DATA_BLOCK "SwitchPLC_Hmi"
{ S7_Optimized_Access := 'TRUE' }
VERSION : 0.1
NON_RETAIN
   VAR RETAIN
      tHMR { ExternalWritable := 'False'} : Struct   // {[Unit]|[Scada Unit]|[LowLimit]|[HigLimit]|[Acces]}
         xCPU1Active { ExternalWritable := 'False'} : Bool;   // Cpu 1 Active {x|x|x|x|O}
         xCPU2Active { ExternalWritable := 'False'} : Bool;   // Cpu 2 Active {x|x|x|x|O}
      END_STRUCT;
   END_VAR


BEGIN

END_DATA_BLOCK

